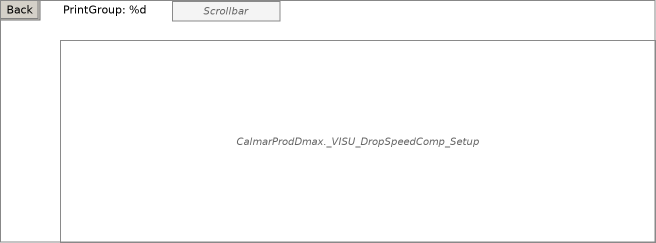
VISUALIZATION VISU_DropSpeedComp_Setup  // 656x243
    Frame (60,40 596x203)
        shows CalmarProdDmax._VISU_DropSpeedComp_Setup(mInst := PRG_PRINT.fbWorkerDefGrid_Print[PRG_PRINT.nVisuSelection_PG].fbDropSpeedComp)
    Button (0,0 40x20), "Back"
        OnMouseClick: change screen: Previous 
    Scrollbar (172,1 108x20)
        p2245068023: iCPr_NB_PG
    Rectangle (60,0 100x20), "PrintGroup: %d", text variable: PRG_PRINT.nVisuSelection_PG
END_VISUALIZATION

(* stored: Version 1.1.0.1, ProductVersion 3.1.4024.11
   Visu VISU_DropSpeedComp_Setup: Id {80422907-1c14-4bcb-86ab-f6aa0e0809fc} *)
